TYPE AxesSetAlphaDeltaVelocityProcessArgs :
STRUCT
	///Units of the alphaVelocity and deltaVelocity
	units: AxesMoveVelocityUnits;
	///Velocity in alpha direction
	alphaVelocity: LREAL;
	///Velocity in delta direction
	deltaVelocity: LREAL;
END_STRUCT
END_TYPE

(* stored: Version 1.1.0.1, ProductVersion 3.1.4019.2
   DUT AxesSetAlphaDeltaVelocityProcessArgs: Id {9d7237f1-846b-4d75-b9e0-566c3f5c3171} *)
